Fanuc KAREL source: kb00152.KL

-- PROVISIONAL review KL for V940-1; original PC SHA256 c82b16996dc098c77695b194fcd612748b10a5ba712632b1620ce061e95bb6a3
-- Incomplete behavior may be omitted. Consult companion uncertainty JSON. Do not deploy.
PROGRAM KB00152
%NOLOCKGROUP
VAR
  P1 : REAL
  RESULT : INTEGER
BEGIN
  -- V9_ZERO_TABLE_METADATA_HINT layout=0001; no indexed target words; source/name/runtime held
  -- UNRESOLVED_PC offsets 5-16; opcodes 2E,23
  -- UNRESOLVED_PC offsets 21-36; opcodes 27,22,76,23
  -- UNRESOLVED_PC offsets 41-45; opcodes 7F
END KB00152
